PROGRAM MAIN
VAR
	ValveController : ValveController;
	InterfaceControlPanel : InterfaceControlPanel;

	StartButton : BOOL;
	ResetButton : BOOL;
	StopButton : BOOL;
	
	StartLight : BOOL;
	ResetLight : BOOL;
	StopLight : BOOL;
	FactoryIOReset: BOOL;

	Setpoint : WORD;
	LevelMeter : WORD;
	
	FillValve : WORD;
	DischargeValve: WORD;
	SP : WORD;
	PV : WORD;
	
	SP_Scaled: REAL;
	LevelScaled: REAL;
	
	isSystemON: BOOL;
	isStopON: BOOL;
	isResetON: BOOL;
	
	tBlink: TON;
	BlinkBit: BOOL;
END_VAR

// I/O Assignments
GVL.mb_Input_Coils[0] := StartLight;
GVL.mb_Input_Coils[1] := ResetLight;
GVL.mb_Input_Coils[2] := StopLight;
GVL.mb_Input_Coils[3] := FactoryIOReset;

StartButton := GVL.mb_Output_Coils[0];
ResetButton := GVL.mb_Output_Coils[1];
StopButton := GVL.mb_Output_Coils[2];

LevelMeter := GVL.mb_Output_Registers[0];
Setpoint := GVL.mb_Output_Registers[2];

GVL.mb_Input_Registers[0] := FillValve;
GVL.mb_Input_Registers[1] := DischargeValve;
GVL.mb_Input_Registers[2] := SP;
GVL.mb_Input_Registers[3] := PV;
//
// Blink bit assignment
tBlink(IN := NOT tBlink.Q, PT := T#1000MS);
BlinkBit := tBlink.ET > T#500MS;
//
// Buttons control initialization
InterfaceControlPanel(StartButton := StartButton, ResetButton := ResetButton, StopButton := StopButton, blink := BlinkBit,
	isStopON := isStopON, isSystemON := isSystemON, isResetON := isResetON, StartLight => StartLight, StopLight => StopLight, ResetLight => ResetLight);
//
// Reset logic
IF ResetButton THEN
	FactoryIOReset := TRUE;
	isSystemON := FALSE;
	isStopON := TRUE;
ELSE
	FactoryIOReset := FALSE;
END_IF;
//
// Setpoint conversion & assignment
AnalogInputConversion(AnalogInput := Setpoint, ScaleMax := 300, ScaledValue => SP_Scaled);
SP := REAL_TO_WORD(SP_Scaled);
//
// Current water level conversion & assignment
AnalogInputConversion(AnalogInput := LevelMeter, ScaleMax := 300, ScaledValue => LevelScaled);
PV := REAL_TO_WORD(LevelScaled);
//
// Valve control logic
IF isSystemON THEN	
	IF PV < SP THEN
		AnalogOutputConversion(0.0, AnalogOutput => DischargeValve);
		ValveController(TargetWaterLevel := SP_Scaled, CurrentWaterLevel := LevelScaled, ScaleMax := 30, AnalogOutputValue => FillValve);
	END_IF;
	IF PV > SP THEN
		AnalogOutputConversion(0.0, AnalogOutput => FillValve);
		ValveController(TargetWaterLevel := LevelScaled, CurrentWaterLevel := SP_Scaled, ScaleMax := 7, AnalogOutputValue => DischargeValve);
	END_IF;
	IF PV = SP THEN
		AnalogOutputConversion(0.0, AnalogOutput => FillValve);
		AnalogOutputConversion(0.0, AnalogOutput => DischargeValve);
	END_IF;
ELSE
	AnalogOutputConversion(0.0, AnalogOutput => FillValve);
	AnalogOutputConversion(0.0, AnalogOutput => DischargeValve);
END_IF;
//

END_PROGRAM

(* stored: Version 1.1.0.1, ProductVersion 3.1.4024.12
   POU MAIN: Id {0e6006db-b60c-47ef-92bd-9d5ed8e74b0e}, SpecialFunc None *)
